TYPE Vec6i : ARRAY[1..6] OF INT; END_TYPE

(* stored: Version 1.1.0.1, ProductVersion 3.1.4024.12
   DUT Vec6i: Id {63465b83-9fa2-4173-a8a4-78896c426934} *)
